INTERFACE IF_Heatpump

METHOD AllowMBComm : BOOL
VAR_INPUT
	b_AllowComm	:	Bool;
END_VAR
END_METHOD

METHOD EMStop : BOOL
VAR_INPUT
END_VAR
END_METHOD

METHOD getDiagnostics
VAR_IN_OUT
	AddError		: ARRAY [*] OF FB_AddErrorST;
	a_ActiveEvents	: ARRAY [*] OF ST_ErrorStruct;
	w_Index			: WORD;
END_VAR

VAR_OUTPUT
	b_errorActive	: BOOL;
	b_warningActive	: BOOL;
END_VAR
END_METHOD

METHOD MBCommBusy : BOOL
VAR_INPUT
END_VAR
END_METHOD

METHOD Reset : BOOL
VAR_INPUT
END_VAR
END_METHOD

METHOD Setpoint : BOOL
VAR_INPUT
	OperatingMode	:	eHeatpumpMode	:= 	eHeatpumpMode.Standby;
	Temperature		: 	REAL			:=	18;
END_VAR
END_METHOD

END_INTERFACE

(* stored: Version 1.1.0.1, ProductVersion 3.1.4024.12
   Itf IF_Heatpump: Id {8df202c4-db2b-4641-abf8-444576336044}
   Method AllowMBComm: Id {9e09d6c9-9f87-44ad-aae9-515ab6ffffa9}
   Method EMStop: Id {bc13dfd9-46d3-401d-988b-0133b3a250c5}
   Method getDiagnostics: Id {aa2107bd-e334-4df5-90ed-4e0e3cc80b9e}
   Method MBCommBusy: Id {926a205b-e3a8-422c-9792-5bb585d58c2e}
   Method Reset: Id {99afb58e-65be-4e86-b507-39090902deed}
   Method Setpoint: Id {d3ad2016-b050-4045-88e7-d909ff27cada} *)
